FUNCTION_BLOCK ACTUATOR
VAR_INPUT
//<!-- PRESPECTIVE_AUTO_INJECT_INPUT_START -->
oToggle : BOOL:= False; //Toggle Bool
//<!-- PRESPECTIVE_AUTO_INJECT_INPUT_END -->
END_VAR
VAR_OUTPUT
//<!-- PRESPECTIVE_AUTO_INJECT_OUTPUT_START -->
iValue : BOOL:= False; //Value
//<!-- PRESPECTIVE_AUTO_INJECT_OUTPUT_END -->
END_VAR
VAR
//<!-- PRESPECTIVE_AUTO_INJECT_VAR_START -->
//<!-- PRESPECTIVE_AUTO_INJECT_VAR_END -->
END_VAR

END_FUNCTION_BLOCK

(* stored: Version 1.1.0.1, ProductVersion 3.1.4022.18
   POU ACTUATOR: Id {7957b515-1401-45d3-bb90-79ecded4fc86}, SpecialFunc None *)
